FUNCTION_BLOCK MainSequencer
VAR_INPUT
	Status	: REFERENCE TO ST_MainSequencerStatus;
END_VAR
VAR
	fbTest1Sequencer	: Test1Sequencer;	
	oPowerPackChargeRequest	 AT%Q* : BOOL;
END_VAR

_M_Test1();
//_M_AutoSequence();

METHOD PRIVATE _M_AutoSequence
VAR_INPUT
END_VAR
fbTest1Sequencer.M_AutoSequence(AutoSteps := E_Test1AutoSteps.PRESSURIZEHYDRAULICMOTOR);
END_METHOD

METHOD PRIVATE _M_Test1
VAR_INPUT
END_VAR
fbTest1Sequencer();
END_METHOD

END_FUNCTION_BLOCK

(* stored: Version 1.1.0.1, ProductVersion 3.1.4024.12
   POU MainSequencer: Id {f7cc08ca-aef1-42fe-82b2-6a0a82031afa}, SpecialFunc None
   Folder Sequence: Id {3289d9b3-554a-4787-becd-9cfb417dba89}
   Method _M_AutoSequence: Id {6cf6cd8d-2e8d-40e2-9a9b-6aba675c9118}
   Method _M_Test1: Id {691a04b7-d6d0-4750-8ccd-7dc021f473b3} *)
